// TIA Portal V18 export
FUNCTION "mot_speed_set_by_lag" : Void   // FC5, FBD
{ S7_Optimized_Access := 'TRUE' }
VERSION : 0.1
// stored: AutoNumber true, IsIECCheckEnabled false, SetENOAutomatically false, UDAEnableTagReadback false
   VAR_INPUT
      SET_SPD : Real;
      MASTER_POS : Real;
      MY_POS : Real;
      par_max_Vcor : Real;
      par_max_Pos_delta : Real;
      parSpeedMinThreshold : Real;
      par_speed_absmax : Real;
      par_dist_absmax : Real;
      par_speed_crawl : Real;
      par_dist_crawl : Real;
      par_dist_stop : Real;
      par_prec_auto : Real;
      isMultiturn : Bool;
      MultiTurnGoesFwdOnly : Bool;
      par_lim_fwd : Real;
      par_lim_rev : Real;
   END_VAR
   VAR_OUTPUT
      SPEED_OUT : Real;
      ER_SET : Bool;
      ER_SET2 : Bool;
      ER_W : WString;
   END_VAR
   VAR_IN_OUT
      should_move : Bool;
   END_VAR
   VAR_TEMP
      delta_pos : Real;
      speed_cor : Real;
      scaled_delta_pos : Real;
      temp_speed : Real;
      speed_target : Real;
      set_speed_substantial : Bool;
      in_vicinity : Bool;
      delta : Real;
      set_speed_miniscule : Bool;
      SET_SPD_ABS : Real;
   END_VAR
BEGIN

REGION Network 1
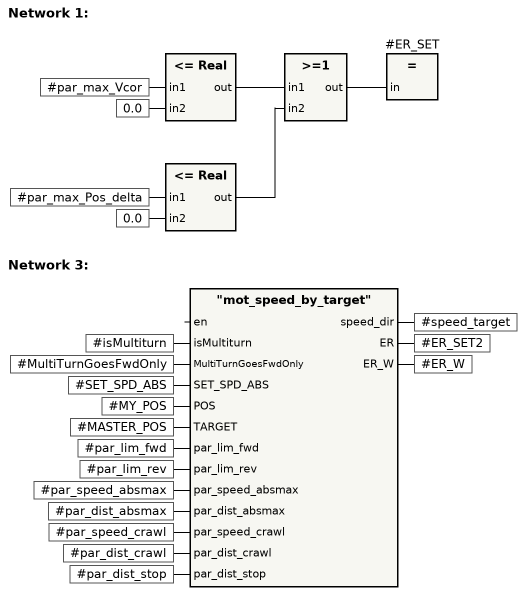
   #ER_SET := (#par_max_Vcor <= 0.0) OR (#par_max_Pos_delta <= 0.0);
END_REGION

REGION Network 2 (SCL)
   #SET_SPD_ABS := ABS(#SET_SPD);
END_REGION

REGION Network 3
   "mot_speed_by_target"(isMultiturn := #isMultiturn,
                         MultiTurnGoesFwdOnly := #MultiTurnGoesFwdOnly,
                         SET_SPD_ABS := #SET_SPD_ABS,
                         POS := #MY_POS,
                         TARGET := #MASTER_POS,
                         par_lim_fwd := #par_lim_fwd,
                         par_lim_rev := #par_lim_rev,
                         par_speed_absmax := #par_speed_absmax,
                         par_dist_absmax := #par_dist_absmax,
                         par_speed_crawl := #par_speed_crawl,
                         par_dist_crawl := #par_dist_crawl,
                         par_dist_stop := #par_dist_stop,
                         speed_dir => #speed_target,
                         ER => #ER_SET2,
                         ER_W => #ER_W);
END_REGION

REGION Network 4 (SCL)
   #delta_pos := LIMIT(IN := #MASTER_POS - #MY_POS, MN := - #par_max_Pos_delta, MX := #par_max_Pos_delta);

   IF (NOT #ER_SET) THEN
       #speed_cor := #par_max_Vcor * #delta_pos / #par_max_Pos_delta;
   ELSE
       #speed_cor := 0;
   END_IF;
END_REGION

REGION Network 5 (SCL)
   #set_speed_substantial := ABS(#SET_SPD) > #parSpeedMinThreshold;
   #set_speed_miniscule := NOT #set_speed_substantial;


   #delta:=ABS(#MY_POS - #MASTER_POS);
   #in_vicinity := #delta < #par_prec_auto;

   IF (#set_speed_substantial) THEN
       #temp_speed := #SET_SPD + #speed_cor;
   ELSE
       #temp_speed := #speed_target;
   END_IF;

   IF #set_speed_substantial OR NOT #in_vicinity THEN
       #should_move := true;
   END_IF;
   IF #set_speed_miniscule AND #speed_target = 0 THEN
       #should_move := false;
   END_IF;


   IF (#should_move) THEN
       #SPEED_OUT := #temp_speed;
   ELSE
       #SPEED_OUT := 0;
   END_IF;
END_REGION
END_FUNCTION
